// TIA Portal V17 export
// export: Created 2022-12-09T10:51:17.483341Z, ExportSetting WithDefaults, DisplayName Totally Integrated Automation Portal, DisplayVersion V17 Update 5, DisplayName TIA Portal Openness, DisplayVersion V17 Update 5, DisplayName TIA Portal Version Control Interface, DisplayVersion V17, DisplayName Simotion SCOUT TIA, DisplayVersion 5.4.3.0, DisplayName SINAMICS Startdrive Advanced, DisplayVersion V17 SP1, DisplayName SINAMICS Startdrive G130, G150, S120, S150, SINAMICS MV, S210, DisplayVersion V17 SP1, DisplayName SINAMICS Startdrive G110M, G120, G120C, G120D, G120P, G115D, DisplayVersion V17 SP1, DisplayName STEP 7 Professional, DisplayVersion V17 Update 5, DisplayName STEP 7 Safety, DisplayVersion V17, DisplayName WinCC Advanced, DisplayVersion V17 Update 5
TYPE "UDT_OMAC_DiagnosticsEntry"
// stored: IsFailsafeCompliant false
   STRUCT
      timestamp : DTL := DTL#1970-01-01-00:00:00;   // Timestamp for this entry
      UnitModeCurrent : Byte := 16#00;   // Current unit mode / Current mode
      StateCurrent : Byte := 16#00;   // Current state
      UnitMode : Byte := 16#00;   // Requested unit mode / Sent Mode
      CntrlCmd : Byte := 16#00;   // Request control command / Sent control command
      SC : Bool := false;   // State complete signal / Sent SC
      message : Byte := 16#00;   // Message for this entry
   END_STRUCT;
END_TYPE
